# EPICS autosave request: iocBoot/tpsCommon.req
$(P):PRESSURE.DESC
$(P):PRESSURE.HIHI
$(P):PRESSURE.HIGH
$(P):PRESSURE.LOW
$(P):PRESSURE.LOLO
$(P):PRESSURE.HHSV
$(P):PRESSURE.HSV
$(P):PRESSURE.LSV
$(P):PRESSURE.LLSV
$(P):PRESSURE.SCAN
